{attribute 'linkalways'} 
{attribute 'no_explicit_call' := 'This FB is a CLASS and must be accessed using methods or properties'}
{attribute 'enable_dynamic_creation'}
FUNCTION_BLOCK Node_F_VN_DrawLinesExp EXTENDS VisionNode
VAR
    ipLines : _ITcVnContainer;
    nLineIndex : _DINT(0);
    ipDestImage : _ITcVnImage;
    aColor : _TcVnVector4_LREAL;
    nThickness : _DINT(1);
    eLineType : _ETcVnLineType(ETcVnLineType.TCVN_LT_4_CONNECTED);
    nShift : _UDINT(0);
    hrPrev : _HRESULT(S_OK);
	hresult : _HRESULT(S_OK);
END_VAR

METHOD PUBLIC  Clone : I_Node
VAR
	pNode : POINTER TO Node_F_VN_DrawLinesExp;
END_VAR
pNode := __NEW(Node_F_VN_DrawLinesExp);
Clone := pNode^;
END_METHOD

METHOD FB_init : BOOL
VAR_INPUT
	bInitRetains : BOOL; // if TRUE, the retain variables are initialized (warm start / cold start)
	bInCopyCode : BOOL;  // if TRUE, the instance afterwards gets moved into the copy code (online change)
END_VAR
AddInput('ipLines', ipLines);
AddParameter('nLineIndex', nLineIndex);
AddInput('ipDestImage', ipDestImage);
AddInput('aColor', aColor);
AddParameter('nThickness', nThickness);
AddParameter('eLineType', eLineType);
AddParameter('nShift', nShift);
AddInput('hrPrev', hrPrev);
AddOutput('ipDestImage', ipDestImage);
AddOutput('hresult',hresult);
END_METHOD

METHOD PROTECTED OnExecute
hresult.Value := F_VN_DrawLinesExp(
    ipLines := ipLines.Value,
    nLineIndex := nLineIndex.Value,
	ipDestImage := ipDestImage.Value,
    aColor := aColor.Value,
    nThickness := nThickness.Value,
    eLineType := eLineType.Value,
    nShift := nShift.Value,
	hrPrev:= hrPrev.Value);
END_METHOD

METHOD PUBLIC PreExecutionCheck
VAR_INPUT
	Check : I_PreExecutionChecks;
END_VAR
Check.IsTrue(ipLines.IsValid, 'ipLines must be a valid container');

Check.IsTrue((ipLines.HasType(TC_GLOBAL_CONST_LIST.ContainerType_Vector_TcVnVector2_REAL) OR
              ipLines.HasType(TC_GLOBAL_CONST_LIST.ContainerType_Vector_TcVnVector4_LREAL) OR
              ipLines.HasType(TC_GLOBAL_CONST_LIST.ContainerType_Vector_TcVnVector4_DINT)),
              'ipLines contains incorrect type');
              
Check.IsTrue(ipDestImage.IsValid, 'ipDestImage must contain an image');
Check.IsTrue(nThickness.Value >= 1, 'nThickness must be greater than or equal to 1');
END_METHOD

END_FUNCTION_BLOCK

(* stored: Version 1.1.0.1, ProductVersion 3.1.4024.15
   POU Node_F_VN_DrawLinesExp: Id {f8504a7a-adc7-0b96-01a0-0ca82cd4a25c}, SpecialFunc None
   Folder Constructor: Id {6742238a-a8c9-0244-2578-40b3446507f5}
   Method Clone: Id {46828fc3-12b8-032f-1df5-7bc16d8a9532}
   Method FB_init: Id {b91a3723-234a-031e-120d-0faff957c7f5}
   Method OnExecute: Id {edd7654a-bfc2-08b0-3605-05e511ff1756}
   Method PreExecutionCheck: Id {328d90f8-2675-0fad-3113-a21c5ad42332} *)
